# EPICS substitutions: ATCACommonApp/Db/StreamFloat.substitutions
file "streamWf.db"  {
    pattern {      PORT,   DEVICE,    WIDTH,  N,   TYPE,                DTYP,      FTVL,       NELM,    TSE      }
            { "$(PORT)", "$(DEV)",  "Float32", 0, "FLOAT", "asynFloat32ArrayOut",   "FLOAT",  "$(NELM\=2048)", "$(TSE)"    }
            { "$(PORT)", "$(DEV)",  "Float32", 1, "FLOAT", "asynFloat32ArrayOut",   "FLOAT",  "$(NELM\=2048)", "$(TSE)"    }
            { "$(PORT)", "$(DEV)",  "Float32", 2, "FLOAT", "asynFloat32ArrayOut",   "FLOAT",  "$(NELM\=2048)", "$(TSE)"    }
            { "$(PORT)", "$(DEV)",  "Float32", 3, "FLOAT", "asynFloat32ArrayOut",   "FLOAT",  "$(NELM\=2048)", "$(TSE)"    }

}
